{attribute 'OPC.UA.DA' := '1'}
{attribute 'OPC.UA.DA.StructuredType' := '1'}
TYPE WavelengthRangeMsg :
STRUCT
	Id : EPowerIlluminationFlow;
	WavelengthRange : STRING(255);
END_STRUCT
END_TYPE

(* stored: Version 1.1.0.1, ProductVersion 3.1.4024.3
   DUT WavelengthRangeMsg: Id {6f67bcd8-ddcb-4bcc-91da-5bce684b8982} *)
